(*			
	RafalOS
	Rafał Osajda		12.11.2025		TC 4024.66
	interfejs potrzebny w HMI
*)
INTERFACE ITF_HMIEMenu_HMI EXTENDS ITF_BaseComponent_HMI

END_INTERFACE

(* stored: Version 1.1.0.1
   Itf ITF_HMIEMenu_HMI: Id {76ad644f-bee1-09cd-13fb-a0a42abb1a07} *)
